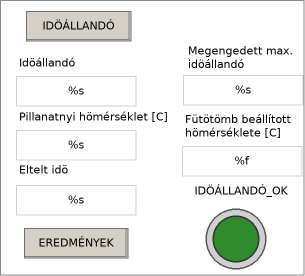
VISUALIZATION Vegmero_idoallando  // 305x276
    Button (26,11 105x30), "IDÖÁLLANDÓ", input disabled if: VEGMERO.s_InCommand<>''
        OnMouseUp: execute { VEGMERO.s_InCommand:='IDOALLANDO'; }
    Textfield (16,76 120x30), "%s", text variable: VEGMERO.tIdoallando
    Textfield (16,130 120x30), "%s", text variable: VEGMERO.arIdoallandoPTTEMP[VEGMERO.nI]
    Textfield (16,185 120x30), "%s", text variable: VEGMERO.atIdoallando[VEGMERO.nI]
    Label (16,53 87x20), "Idöállandó"
    Label (16,107 164x20), "Pillanatnyi hömérséklet [C]"
    Label (16,160 89x20), "Eltelt idö"
    Lamp1 (201,204 70x70), variable: NOT VEGMERO.bIDOALLANDO_OK, style: Lamp-Lamp1-Red
    Label (186,181 110x20), "IDÖÁLLANDÓ_OK"
    Textfield (182,146 120x30), "%f", text variable: GVL.rTempMax
    Label (182,109 117x34), "Fütötömb beállított hömérséklete [C]"
    Textfield (183,75 120x30), "%s", text variable: REAL_TO_TIME(GVL.rIdoallandoMax*1000)
    Label (185,43 107x29), "Megengedett max. idöállandó"
    Lamp1 (201,204 70x70), variable: VEGMERO.bIDOALLANDO_OK, invisible if: NOT VEGMERO.bIDOALLANDO_OK AND VEGMERO.bIDOALLANDO_MERVE, style: Lamp-Lamp1-Green
    Button (24,228 104x30), "EREDMÉNYEK"
        OnMouseUp: execute { GVL.bMeresiEredmenyekRejtve:=FALSE; }
END_VISUALIZATION

(* stored: Version 1.1.0.1, ProductVersion 3.1.4024.11
   Visu Vegmero_idoallando: Id {017539d3-0418-4feb-b40e-6b79a157cd54} *)
